                             //Check Subscribe ACK paket
                             CASE #tempMqttSubAckRcv OF
                               #NO_RESPONSE:  // Statement section case 1
                                 ;
                               #RESPONSE_GOOD:  // Statement section case 2 to 4
                                 //disable watchdog
                                 #statEnableTimerCommandWatchdog := FALSE;
                                 //Encoding done all sent
                                 #statPaketHeaderEncodeDone := FALSE;
                                 // Job done
                                 #statDone := TRUE;
                                 #statMqttCommandState := #MQTT_COMMAND_STATE_NO_PROCESSING;
                                 // Set Status back to connected
                                 #statStatus := #STATUS_JOB_EXECUTED;
                               #RESPONSE_PAKET_ID_INVALID:  // PaketId Invalid
                                 #statStatus := #ERR_MQTT_PAKET_ID_INVALID; // Set correct status that identifies error clearly
                                 #statSubfunctionStatus := #ERR_MQTT_PAKET_ID_INVALID; // Status or return value of called FBs, FCs and system blocks
                                 #statFBErrorState := #statFBState; // Set error state number for diagnostic 
                                 #statErrorAutoCleared := TRUE;
                                 #statMqttCommandState := #MQTT_COMMAND_STATE_NO_PROCESSING;
                               #RESPONSE_SUBSCRIBE_FAILED:
                                 #statStatus := #ERR_MQTT_SUBACK_FAILURE; // Set correct status that identifies error clearly
                                 #statSubfunctionStatus := #ERR_MQTT_SUBACK_FAILURE; // Status or return value of called FBs, FCs and system blocks
                                 #statFBErrorState := #statFBState; // Set error state number for diagnostic 
                                 #statErrorAutoCleared := TRUE;
                                 #statMqttCommandState := #MQTT_COMMAND_STATE_NO_PROCESSING;
                             END_CASE;
                           END_REGION SEND_SUBSCRIBE_WAIT_FOR_RESPONSE

                         #MQTT_COMMAND_STATE_BUILD_UNSUBSCRIBE:// Unsubscribe from topics
                           REGION UNSUBSCRIBE_FROM_TOPIC
                             //Remaining Length is the length of the variable header (PacketID, 2Bytes) plus the length of the Payload. 
                             //Max Len of Mqtt pakets is per Standard 268,435,455 Bytes (ff,ff,ff,7f)
                             //Calculate Remain Len will be
                             //Len of TOPIC   (max 3*16382 WChars= 49.146 Bytes)
                             //LenInfo Topic (2Byte)
                             //
                             //Set Status
                             #statStatus := #STATUS_MQTT_UNSUBSCRIBE;
                             // Must obey, if not currently sending PubAck Msg on a subscription
                             // Else, try in the next cycle
                             IF #tempTsendcBusy = FALSE // when tsendC is ready
                               AND #tempTsendcDone = FALSE // tsendC did not finish in this cycle
                               AND #statTsendcReq = FALSE // TsendC request was not already requested by pub ack msg
                             THEN
                               //Header not encoded
                               IF #statPaketHeaderEncodeDone = FALSE THEN
                                 //Init
                                 #statSendPaketTotalRemLen := 0;
                                 #statSendBufferPos := 0;
                                 #statUnsubscribeTopicEncodeState := #FIRST_ENCODING;
                                 #statUnsubscribeTopicPos := #FIRST_CHARACTER;
                                 #statUnsubscribeTopicLenUtf8Encoded := 0;
                                 #statPaketId += 1;//increment

                                 //check necessary boundaries

                                 IF LEN(#mqttTopic) = #LEN_NULL THEN
                                   #statStatus := #ERR_MQTT_COMMAND_UNSUBSCRIBE_TOPIC_INVALID; // Set correct status that identifies error clearly
                                   #statSubfunctionStatus := #ERR_MQTT_COMMAND_UNSUBSCRIBE_TOPIC_INVALID; // Status or return value of called FBs, FCs and system blocks
                                   #statFBErrorState := #statFBState; // Set error state number for diagnostic 
                                   #statErrorUserCleared := TRUE;
                                 ELSE // All ok
                                   //Add two Byte for Paket ID:
                                   #statSendPaketTotalRemLen := #statSendPaketTotalRemLen + #TWO_BYTE_LEN_INFO;
                                   //add unsubscribe  topic len
                                   FOR #tempLoopCounter := #FIRST_CHARACTER TO LEN(#mqttTopic) DO
                                     "LMQTT_ConvertToUtf8"(character     := #mqttTopic[#tempLoopCounter],
                                                           convertedUtf8 => #tempConvertedUtf8,
                                                           bytesUsed     => #tempBytesUsedUtf8,
                                                           error         => #tempErrorConvertUtf8,
                                                           status        => #tempStatusConvertUtf8);
                                     #statUnsubscribeTopicLenUtf8Encoded := #statUnsubscribeTopicLenUtf8Encoded + #tempBytesUsedUtf8;
                                   END_FOR;
                                   //Add len of topic plus len info
                                   #statSendPaketTotalRemLen := #statSendPaketTotalRemLen + #statUnsubscribeTopicLenUtf8Encoded + #TWO_BYTE_LEN_INFO;

                                   //Build Subscribe Telegram
                                   //Fixed Header - Write Paket Type
                                   #statSendBuffer[#statSendBufferPos] := #MQTT_MSG_TYPE_UNSUBSCRIBE;
                                   #statSendBufferPos += 1; // increment

                                   //Write Remaining Paket Len info 
                                   WHILE (#statSendPaketTotalRemLen > #DEFAULT_VALUE_ZERO)
                                   DO//See MQTT Spec for explanation of this calculation
                                     #statEncodedRemPaketLenAsByte := UDINT_TO_BYTE(#statSendPaketTotalRemLen MOD #SEND_LEN_MULTIPLIER_UDINT_128);
                                     #statSendPaketTotalRemLen := #statSendPaketTotalRemLen / #SEND_LEN_MULTIPLIER_UDINT_128;
                                     // if there are more data to encode, set the top bit of this byte
                                     IF #statSendPaketTotalRemLen > #DEFAULT_VALUE_ZERO
                                     THEN
                                       // Do this and continue while loop
                                       #statEncodedRemPaketLenAsByte := #statEncodedRemPaketLenAsByte OR UDINT_TO_BYTE(#SEND_LEN_MULTIPLIER_UDINT_128);
                                       #statSendBuffer[#statSendBufferPos] := #statEncodedRemPaketLenAsByte;
                                       #statSendBufferPos += 1;
                                     ELSE
                                       //do this and leave while loop
                                       #statSendBuffer[#statSendBufferPos] := #statEncodedRemPaketLenAsByte;
                                       #statSendBufferPos += 1;
                                     END_IF;
                                   END_WHILE;

                                   // Set Paket Id
                                   #tempWordForSliceAddress := UINT_TO_WORD(#statPaketId);
                                   #statSendBuffer[#statSendBufferPos] := #tempWordForSliceAddress.%B1; //MSB
                                   #statSendBufferPos += 1;
                                   #statSendBuffer[#statSendBufferPos] := #tempWordForSliceAddress.%B0; //LSB
                                   #statSendBufferPos += 1;

                                   //When all done, set encode to true
                                   #statPaketHeaderEncodeDone := TRUE;
                                 END_IF;
                               END_IF;

                               //Header Encoded - 
                               IF #statPaketHeaderEncodeDone = TRUE THEN
                                 //Unsubscribe Topic
                                 IF #statSendBufferPos <= #MAX_BUFFER_LEN_SEND - #TWO_BYTE_LEN_INFO THEN
                                   CASE #statUnsubscribeTopicEncodeState OF
                                     #FIRST_ENCODING:  // Statement section case 1
                                       //ADD len info into paket

                                       #tempWordForSliceAddress := UINT_TO_WORD(#statUnsubscribeTopicLenUtf8Encoded);
                                       #statSendBuffer[#statSendBufferPos] := #tempWordForSliceAddress.%B1; //MSB
                                       #statSendBufferPos += 1;
                                       #statSendBuffer[#statSendBufferPos] := #tempWordForSliceAddress.%B0; // LSB
                                       #statSendBufferPos += 1;

                                       FOR #tempLoopCounter := #statUnsubscribeTopicPos TO LEN(#mqttTopic) DO
                                         "LMQTT_ConvertToUtf8"(character     := #mqttTopic[#tempLoopCounter],
                                                               convertedUtf8 => #tempConvertedUtf8,
                                                               bytesUsed     => #tempBytesUsedUtf8,
                                                               error         => #tempErrorConvertUtf8,
                                                               status        => #tempStatusConvertUtf8);

                                         IF #statSendBufferPos + #tempBytesUsedUtf8 <= #MAX_BUFFER_LEN_SEND THEN
                                           #statUnsubscribeTopicPos += 1;
                                           CASE #tempBytesUsedUtf8 OF
                                             #UTF_1_BYTE_USED:  // Statement section case 1
                                               #statSendBuffer[#statSendBufferPos] := #tempConvertedUtf8.%B0;
                                               #statSendBufferPos += 1;
                                             #UTF_2_BYTE_USED:
                                               #statSendBuffer[#statSendBufferPos] := #tempConvertedUtf8.%B0;
                                               #statSendBufferPos += 1;
                                               #statSendBuffer[#statSendBufferPos] := #tempConvertedUtf8.%B1;
                                               #statSendBufferPos += 1;
                                             #UTF_3_BYTE_USED:  // Statement section case 2 to 4
                                               #statSendBuffer[#statSendBufferPos] := #tempConvertedUtf8.%B0;
                                               #statSendBufferPos += 1;
                                               #statSendBuffer[#statSendBufferPos] := #tempConvertedUtf8.%B1;
                                               #statSendBufferPos += 1;
                                               #statSendBuffer[#statSendBufferPos] := #tempConvertedUtf8.%B2;
                                               #statSendBufferPos += 1;
                                             ELSE  // Statement section ELSE
                                               ;
                                           END_CASE;
                                         ELSE
                                           //When buffer full
                                           #statUnsubscribeTopicEncodeState := #SUBSEQUENT_ENCODING;
                                           EXIT;
                                         END_IF;
                                       END_FOR;
                                       IF #statUnsubscribeTopicPos >= LEN(#mqttTopic) THEN
                                         #statUnsubscribeTopicEncodeState := #ENCODE_DONE;
                                       END_IF;

                                     #SUBSEQUENT_ENCODING:  // Statement section case 2 to 4
                                       FOR #tempLoopCounter := #statUnsubscribeTopicPos TO LEN(#mqttTopic) DO

                                         "LMQTT_ConvertToUtf8"(character     := #mqttTopic[#tempLoopCounter],
                                                               convertedUtf8 => #tempConvertedUtf8,
                                                               bytesUsed     => #tempBytesUsedUtf8,
                                                               error         => #tempErrorConvertUtf8,
                                                               status        => #tempStatusConvertUtf8);
                                         IF #statSendBufferPos + #tempBytesUsedUtf8 <= #MAX_BUFFER_LEN_SEND THEN
                                           #statUnsubscribeTopicPos += 1;
                                           CASE #tempBytesUsedUtf8 OF
                                             #UTF_1_BYTE_USED:  // Statement section case 1
                                               #statSendBuffer[#statSendBufferPos] := #tempConvertedUtf8.%B0;
                                               #statSendBufferPos += 1;
                                             #UTF_2_BYTE_USED:
                                               #statSendBuffer[#statSendBufferPos] := #tempConvertedUtf8.%B0;
                                               #statSendBufferPos += 1;
                                               #statSendBuffer[#statSendBufferPos] := #tempConvertedUtf8.%B1;
                                               #statSendBufferPos += 1;
                                             #UTF_3_BYTE_USED:  // Statement section case 2 to 4
                                               #statSendBuffer[#statSendBufferPos] := #tempConvertedUtf8.%B0;
                                               #statSendBufferPos += 1;
                                               #statSendBuffer[#statSendBufferPos] := #tempConvertedUtf8.%B1;
                                               #statSendBufferPos += 1;
                                               #statSendBuffer[#statSendBufferPos] := #tempConvertedUtf8.%B2;
                                               #statSendBufferPos += 1;
                                             ELSE  // Statement section ELSE
                                               ;
                                           END_CASE;
                                         ELSE
                                           //When buffer full
                                           EXIT;
                                         END_IF;
                                       END_FOR;
                                       IF #statUnsubscribeTopicPos >= LEN(#mqttTopic) THEN
                                         #statUnsubscribeTopicEncodeState := #ENCODE_DONE;
                                       END_IF;
                                     ELSE  // Skip when Done
                                       ;
                                   END_CASE;
                                 END_IF;

                                 //set Sendlen for TSendC Block
                                 #statTsendcLen := #statSendBufferPos; // Buffer pos equals amount of elements in send array
                                 //reset buffer pos
                                 #statSendBufferPos := 0;
                                 //enable Send Req
                                 #statTsendcReq := TRUE;
                                 //Set Watchdog
                                 #statEnableTimerCommandWatchdog := TRUE;
                                 //wait for send to be done
                                 #statMqttCommandState := #MQTT_COMMAND_STATE_SEND_UNSUBSCRIBE;
                               END_IF;
                             END_IF;
                           END_REGION UNSUBSCRIBE_FROM_TOPIC

                         #MQTT_COMMAND_STATE_SEND_UNSUBSCRIBE:
                           REGION SEND_UNSUBSCRIBE_WAIT_FOR_RESPONSE
                             //check tsend status
                             IF NOT #tempTsendcBusy AND #tempTsendcStatus = #TSENDC_JOB_DONE THEN
                               IF (#statUnsubscribeTopicEncodeState = #ENCODE_DONE) THEN
                                 //Encoding done all sent
                                 #statPaketHeaderEncodeDone := FALSE;
                               ELSE
                                 // More to Encode and send
                                 #statEnableTimerCommandWatchdog := FALSE;
                                 #statMqttCommandState := #MQTT_COMMAND_STATE_BUILD_UNSUBSCRIBE;
                               END_IF;
                             END_IF;
                             // Wait for timeout
                             IF #instTimerCommandWatchdog.Q THEN
                               #statEnableTimerCommandWatchdog := FALSE;
                               #statStatus := #ERR_MQTT_COMMAND_SEND_TIMEOUT; // Set correct status that identifies error clearly
                               #statSubfunctionStatus := #ERR_MQTT_COMMAND_SEND_TIMEOUT; // Status or return value of called FBs, FCs and system blocks
                               #statFBErrorState := #statFBState; // Set error state number for diagnostic 
                               #statErrorAutoCleared := TRUE;
                               #statMqttCommandState := #MQTT_COMMAND_STATE_NO_PROCESSING;
                             END_IF;
                             //Check Unsubscribe ACK paket
                             CASE #tempMqttUnSubAckRcv OF
                               #NO_RESPONSE:  // Statement section case 1
                                 ;
                               #RESPONSE_GOOD:  // Statement section case 2 to 4
                                 //disable watchdog
                                 #statEnableTimerCommandWatchdog := FALSE;
                                 //Encoding done all sent
                                 #statPaketHeaderEncodeDone := FALSE;
                                 // Job done
                                 #statDone := TRUE;
                                 #statMqttCommandState := #MQTT_COMMAND_STATE_NO_PROCESSING;
                                 // Set Status back to connected
                                 #statStatus := #STATUS_JOB_EXECUTED;
                               #RESPONSE_PAKET_ID_INVALID:
                                 #statStatus := #ERR_MQTT_PAKET_ID_INVALID; // Set correct status that identifies error clearly
                                 #statSubfunctionStatus := #ERR_MQTT_PAKET_ID_INVALID; // Status or return value of called FBs, FCs and system blocks
                                 #statFBErrorState := #statFBState; // Set error state number for diagnostic 
                                 #statErrorAutoCleared := TRUE;
                                 #statMqttCommandState := #MQTT_COMMAND_STATE_NO_PROCESSING;
                             END_CASE;
                           END_REGION SEND_UNSUBSCRIBE_WAIT_FOR_RESPONSE

                         #MQTT_COMMAND_STATE_SEND_PING:
                           REGION SEND_PING
                             //Set Status
                             #statStatus := #STATUS_MQTT_PING;
                             IF #tempTsendcBusy = FALSE // when tsendC is ready
                               AND #tempTsendcDone = FALSE // tsendC did not finish in this cycle
                               AND #statTsendcReq = FALSE // TsendC request was not already requested by pub ack msg
                             THEN
                               //Init
                               #statSendBufferPos := 0;
                               #statSendBuffer[#statSendBufferPos] := #MQTT_MSG_TYPE_PING;
                               #statSendBufferPos += 1;
                               //Remaining Lenght (must be 0)
                               #statSendBuffer[#statSendBufferPos] := 0;
                               #statSendBufferPos += 1;
                               #statTsendcLen := #statSendBufferPos;
                               //Start send request
                               #statTsendcReq := TRUE;
                               //Start watchdoc
                               #statEnableTimerCommandWatchdog := true;
                               //Next state
                               #statMqttCommandState := #MQTT_COMMAND_STATE_PING_RESP;
                             END_IF;
                           END_REGION MQTT_COMMAND_SEND_PING

                         #MQTT_COMMAND_STATE_PING_RESP:
                           REGION WAIT_FOR_PING_RESP
                             //Check, if Edge of Publish comes while ping
                             IF #tempCommandInput > 0 AND NOT #statCommandInputOld THEN
                               #statCommandInputBackup := #tempCommandInput;
                               #statCommandInputOld := true;
                             END_IF;
                             //check watchdog status
                             IF #instTimerCommandWatchdog.Q THEN
                               #statEnableTimerCommandWatchdog := FALSE;
                               #statStatus := #ERR_MQTT_COMMAND_SEND_TIMEOUT; // Set correct status that identifies error clearly
                               #statSubfunctionStatus := #ERR_MQTT_COMMAND_SEND_TIMEOUT; // Status or return value of called FBs, FCs and system blocks
                               #statFBErrorState := #statFBState; // Set error state number for diagnostic 
                               #statErrorAutoCleared := TRUE;
                               #statMqttCommandState := #MQTT_COMMAND_STATE_NO_PROCESSING;
                             END_IF;
                             //Check PingRsp paket
                             CASE #tempMqttPingRspRcv OF
                               #NO_RESPONSE:  // Statement section case 1
                                 ;
                               #RESPONSE_GOOD:
                                 //disable watchdog
                                 #statEnableTimerCommandWatchdog := FALSE;
                                 //Go to no processing
                                 #statMqttCommandState := #MQTT_COMMAND_STATE_NO_PROCESSING;
                                 //set Status
                                 #statStatus := #STATUS_MQTT_CONNECTED;
                                 IF #statCommandInputBackup <> 0 THEN
                                   #statMqttCommandState := BYTE_TO_DINT(#statCommandInputBackup);
                                   #statCommandInputBackup := 0;
                                   #statCommandInputOld := false;
                                 END_IF;
                             END_CASE;
                           END_REGION MQTT_COMMAND_PING_RESP
                         ELSE  // Statement section ELSE
                           REGION ERROR_MULTIPLE_INPUT
                             #statMqttCommandState := #MQTT_COMMAND_STATE_NO_PROCESSING; // reset back to idle
                             #statStatus := #ERR_MQTT_COMMAND_MULTIPLE_INPUT; // Set correct status that identifies error clearly
                             #statSubfunctionStatus := #ERR_MQTT_COMMAND_MULTIPLE_INPUT; // Status or return value of called FBs, FCs and system blocks
                             #statFBErrorState := #statFBState; // Set error state number for diagnostic 
                             #statErrorAutoCleared := TRUE;
                           END_REGION ERROR_MULTIPLE_INPUT 
                       END_CASE;
                     END_REGION

                     REGION CHECK_PING_TIMER
                       //If no job is running check if keepalive experied
                       IF #statMqttCommandState = #MQTT_COMMAND_STATE_NO_PROCESSING
                         AND #instMqttKeepAliveTimer.Q THEN
                         //reset the timer
                         RESET_TIMER(#instMqttKeepAliveTimer);
                         //go to ping state
                         #statMqttCommandState := #MQTT_COMMAND_STATE_SEND_PING;
                       END_IF;
                     END_REGION CHECK_PING_TIMER

                     //Edge detection "publish / subscribe/unsubscribe" input
                     #statPublishOld := #tempPublish;
                     #statSubscribeOld := #tempSubscribe;
                     #statUnsubscribeOld := #tempUnsubscribe;
                   END_REGION CONNECTED

                 ELSE   // Undefined state in state machine reached
                   #statStatus := #ERR_UNDEFINED_STATE;
                   #statErrorUserCleared := TRUE;
               END_CASE;

             END_REGION MQTT_STATE_MACHINE
           END_IF;
         END_REGION FB_OPERATING_MONITOR_TCP

       #FB_STATE_TCP_RECONNECTING:
         REGION FB_STATE_TCP_RECONNECTING
           IF #tempTsendcStatus = #TSENDC_EST_OK THEN
             #statErrorAutoCleared := FALSE;
             // Update edge detection
             #statPublishOld := #tempPublish;
             #statSubscribeOld := #tempSubscribe;
             #statUnsubscribeOld := #tempUnsubscribe;
             //Monitor Connection
             #statFBState := #FB_STATE_OPERATING_MONITOR_TCP;
             // Begin MQTT Connection
             #statMqttConnectState := #MQTT_CONNECT_STATE_BUILD_PAKET;
           END_IF;
         END_REGION FB_STATE_TCP_RECONNECTING
       #FB_STATE_DISABLING: // Disabling active
         REGION DISABLING FB
           //  Disabling, e.g. closing connections, etc.
           // When disabling is complete the bit #statDisablingCompleted must be set
           // When MQTT is connected, send disconnect
           IF #statMqttConnectState = #MQTT_CONNECT_STATE_CONNECTED THEN
             IF #statTsendcReq = TRUE THEN
               //Interrupt any existing send jobs
               #statTsendcReq := FALSE;
             ELSE
               // INIT
               #statSendBufferPos := 0;
               //Build fixed Header
               //Message Type
               #statSendBuffer[#statSendBufferPos] := #MQTT_MSG_TYPE_DISCONNECT;
               #statSendBufferPos += 1;
               //Remaining Length (must be O)
               #statSendBuffer[#statSendBufferPos] := #REMAINIG_LEN_0;
               #statSendBufferPos += 1;
               //send request
               #statTsendcLen := #statSendBufferPos;
               #statTsendcReq := TRUE;
               #statMqttConnectState := #MQTT_CONNECT_STATE_DISCONNECTED;
             END_IF;
           ELSE
             //Disable TCP Connection
             #statTsendcReq := FALSE;
             #statTsendcEnable := FALSE;
             #statEnableTimerCommandWatchdog := TRUE;
           END_IF;
           // When TCP connection is closed
           IF #tempTsendcStatus = #TSENDC_DISCONNECTED THEN
             #statEnableTimerCommandWatchdog := FALSE;
             #statDisablingCompleted := TRUE;
           ELSIF #instTimerCommandWatchdog.Q THEN
             #statEnableTimerCommandWatchdog := FALSE;
             #statDisablingCompleted := TRUE;
           END_IF;
         END_REGION DISABLING FB
       ELSE // Undefined state in state machine reached
         #statStatus := #ERR_UNDEFINED_STATE;
         #statErrorUserCleared := TRUE;
     END_CASE;
   END_REGION STATE_MACHINE

   REGION OUTPUTS
     // Write outputs
     IF (#statDisablingCompleted = TRUE) THEN
       // Reset outputs if disabling completed
       #statValid := FALSE;
       #statBusy := FALSE;
       #statError := FALSE;
       #statDone := FALSE;
       #statErrorUserCleared := FALSE;
       #statErrorAutoCleared := FALSE;
       #statStatus := #STATUS_NO_CALL;
       // Reset application specific outputs
       #statRcvMsgStatus := #MSG_DECODE_STATUS_NO_NEW_MSG;
       #statRcvMsgDataLen := 0;

     ELSIF (#statErrorUserCleared = TRUE) AND (#statError = FALSE) THEN
       // Error can only be cleared by user; rising edge at enable input is needed to continue 
       #statValid := FALSE;
       #statBusy := FALSE;
       #statDone := FALSE;
       #statError := TRUE;
       // Write diagnostics
       #diagnostics.status := #statStatus;
       #diagnostics.subfunctionStatus := #statSubfunctionStatus;
       #diagnostics.stateNumber := #statFBErrorState;
       // execution aborted --> set state no processing
       #statTsendcEnable := FALSE; // Terminate Connection, no reason keep it up.
       #statFBState := #FB_STATE_NO_PROCESSING;
       #statMqttConnectState := #MQTT_CONNECT_STATE_NO_PROCESSING;
       #statMqttCommandState := #MQTT_COMMAND_STATE_NO_PROCESSING;
       #statRcvMsgDecodeState := #MSG_DECODE_STATE_NO_PROCESSING;

     ELSIF (#statErrorAutoCleared = TRUE) AND (#statError = FALSE) THEN
       // Error can be reset by FB automatically
       #statValid := FALSE;
       #statBusy := TRUE;
       #statError := TRUE;
       #statDone := FALSE;

       // Write diagnostics
       #diagnostics.status := #statStatus;
       #diagnostics.subfunctionStatus := #statSubfunctionStatus;
       #diagnostics.stateNumber := #statFBErrorState;
       // Handling of autocleared error
       CASE #statStatus OF
           //Just signal error and reset autocleared error afterwards.
         #ERR_MQTT_PAKET_ID_INVALID, #ERR_MQTT_SUBACK_FAILURE, #ERR_MQTT_CONNECT_TIMEOUT,
         #ERR_MQTT_COMMAND_SEND_TIMEOUT, #ERR_MQTT_COMMAND_MULTIPLE_INPUT, #ERR_CNT_EXCEEDS_ARRAY_DIMENSION,
         #ERR_MQTT_COMMAND_PUBLISH_TOPIC_INVALID, #ERR_QOS_INVALID, #ERR_MQTT_COMMAND_SUBSCRIBE_TOPIC_INVALID:
           #statErrorAutoCleared := FALSE;

         ELSE  // Statement section ELSE
           ;
       END_CASE;

     ELSIF (#statErrorAutoCleared = FALSE) AND (#statErrorUserCleared = FALSE) AND (#statError = TRUE) THEN
       // If autocleared error is acknowledged
       #statValid := TRUE;
       #statBusy := TRUE;
       #statError := FALSE;
       #statDone := FALSE;

       //   this line  more detailed status information is used instead of "#STATUS_SUBSEQUENT_CALL"
       CASE #statStatus OF
         #ERR_TCP_RECONNECTING, #ERR_MQTT_CONNECT_TIMEOUT:  // Reconnecting ok, start Mqtt reconnnect
           //set status
           #statStatus := #STATUS_MQTT_CONNECTING;
           //in the following status codes status stays connected. 
         #ERR_MQTT_PAKET_ID_INVALID, #ERR_MQTT_SUBACK_FAILURE, #ERR_MQTT_COMMAND_SEND_TIMEOUT,
         #ERR_MQTT_COMMAND_MULTIPLE_INPUT, #ERR_CNT_EXCEEDS_ARRAY_DIMENSION, #ERR_MQTT_COMMAND_PUBLISH_TOPIC_INVALID,
         #ERR_QOS_INVALID, #ERR_MQTT_COMMAND_SUBSCRIBE_TOPIC_INVALID:
           #statStatus := #STATUS_MQTT_CONNECTED;
         ELSE  // Statement section ELSE
           ;
       END_CASE;
     END_IF;

     // Write static values to outputs
     #valid := #statValid;
     #busy := #statBusy;
     #error := #statError;
     #status := #statStatus;
     //block sets ENO automatically:
     //ENO := TRUE;
     //Write application specific static values to outputs
     #done := #statDone;
     #receivedMsgStatus := #statRcvMsgStatus;
     #receivedMsgDataLen := #statRcvMsgDataLen;
   END_REGION OUTPUTS
END_FUNCTION_BLOCK

// folder: LMQTT/Utilities

FUNCTION "LMQTT_ConvertToUtf8" : Void   // FC6, SCL
TITLE = LMQTT_ConvertToUtf8
{ S7_Optimized_Access := 'TRUE' }
AUTHOR : SIEMENS
FAMILY : LMQTT
VERSION : 1.0
// Function to convert a WCHAR to a UTF-8 conformant byte sequence
   VAR_INPUT
      character : WChar;   // Character that shall be converted to UTF-8
   END_VAR
   VAR_OUTPUT
      convertedUtf8 : DWord;   // UTF-8 conformant byte sequence. B0 stores first Byte, B1 second and B2 third Byte. B3 is not used
      bytesUsed : USInt;   // Amount of Bytes converted. Ranges from 1 to 3.
      error : Bool;   // TRUE: An error occurred during the execution of the FC
      status : Word;   // 16#0000 - 16#7FFF: Status of the FC, 16#8000 - 16#FFFF: Error identification
   END_VAR
   VAR_TEMP
      tempStatus : Word;   // temp value for output 'status'
      tempConvertedUtf8 : DWord;   // temp value for output 'convertedUtf8'
      tempBytesUsed : USInt;   // temp value for output 'bytesUsed'
      tempCharacter : WChar;   // temp value for input 'character'
   END_VAR
   // Ret_Val : No return for this FC - see error and status output
   VAR CONSTANT
      STATUS_NO_ERROR : Word := 16#0000;   // no error status
      STATUS_EXECUTION_FINISHED : Word := 16#0000;   // Execution finished without errors
      ERR_UNDEFINED : Word := 16#8000;   // Error due to an undefined case
      USINT_NULL : USInt := 0;   // Init value with 0
      DWORD_NULL : DWord := 16#0000_0000;   // Init value with 0
      EMPTY_WCHAR : WChar := WCHAR#' ';   // Empty WChar for comparison
      BELOW_7F : Word := 16#007F;   // Upper limit for character if only one Byte used
      BELOW_7FF : Word := 16#07FF;   // Upper limit for character if two Byte used
      BELOW_MAX_FFFF : Word := 16#FFFF;   // Upper limit for character if three Byte used
      BYTE_3F : Byte := 16#3F;   // Conversion Value
      BYTE_80 : Byte := 16#80;   // Conversion Value
      BYTE_C0 : Byte := 16#C0;   // Conversion Value
      BYTE_E0 : Byte := 16#E0;   // Conversion Value
      USINT_ONE : USInt := 1;   // Const Value to assign amount of bytes used
      USINT_TWO : USInt := 2;   // Const Value to assign amount of bytes used
      USINT_THREE : USInt := 3;   // Const Value to assign amount of bytes used
   END_VAR
BEGIN
   REGION BLOCK INFO HEADER
       //=============================================================================
       // SIEMENS AG
       // (c)Copyright 2020
       //-----------------------------------------------------------------------------
       // Library:       LMQTT
       // Tested with:   CPU 1516-3 PN/DP V2.8
       // Engineering:   TIA Portal V16
       // Restrictions:  --
       // Requirements:  --
       // Functionality: Converts a single WChar Character to a valid UTF-8 encoded byte sequence and saves this to a DWord.
       //                The amount of bytes saved is stored in bytesUsed Output.
       //-----------------------------------------------------------------------------
       // Change log table:
       // Version    Date         Expert in charge         Changes applied
       // 03.00.00   01.10.2020   Siemens Online Support   First released version
       //=============================================================================
   END_REGION

   REGION INITIALISATION  
       // Initialize functionality: reset of variables, diagnostics, etc.
       #tempConvertedUtf8 := #DWORD_NULL;
       #tempBytesUsed := #USINT_NULL;
       #tempStatus := #STATUS_NO_ERROR;
       //assign temp value from input:
        #tempCharacter := #character;

   END_REGION

   REGION PROGRAM LOGIC
       // Use this region for application specific code
       IF #tempCharacter = #EMPTY_WCHAR THEN
           //will be only 1 byte occupied
           #tempConvertedUtf8 := WCHAR_TO_DWORD(#tempCharacter);
           #tempBytesUsed := #USINT_ONE;
       ELSIF (WCHAR_TO_WORD(#tempCharacter) <= (#BELOW_7F)) THEN
           //will be only 1 byte occupied
           #tempConvertedUtf8 := WCHAR_TO_DWORD(#tempCharacter);
           #tempBytesUsed := #USINT_ONE;
       ELSIF (WCHAR_TO_WORD(#tempCharacter) <= (#BELOW_7FF)) THEN
           //will be 2 byte occupied
           #tempConvertedUtf8.%B1 := (WCHAR_TO_BYTE(#tempCharacter) AND #BYTE_3F) OR #BYTE_80;
           #tempConvertedUtf8.%B0 := WORD_TO_BYTE(SHR(IN := WCHAR_TO_WORD(#tempCharacter), N := 6)) OR #BYTE_C0;
           #tempBytesUsed := #USINT_TWO;
       ELSIF (WCHAR_TO_WORD(#tempCharacter) <= (#BELOW_MAX_FFFF)) THEN
           //will be 3 byte occupied
           #tempConvertedUtf8.%B2 := (WCHAR_TO_BYTE(#tempCharacter) AND #BYTE_3F) OR #BYTE_80;
           #tempConvertedUtf8.%B1 := (WORD_TO_BYTE(SHR(IN := WCHAR_TO_WORD(#tempCharacter), N := 6)) AND #BYTE_3F) OR #BYTE_80;
           #tempConvertedUtf8.%B0 := WORD_TO_BYTE(SHR(IN := WCHAR_TO_WORD(#tempCharacter), N := 12)) OR #BYTE_E0;
           #tempBytesUsed := #USINT_THREE;
       END_IF;
   END_REGION

   REGION OUTPUTS
       // Write application specific temp values to outputs
       #bytesUsed := #tempBytesUsed;
       #convertedUtf8 := #tempConvertedUtf8;
       // Write error and status
       #error := #tempStatus.%X15;
       #status := #tempStatus;
       // ENO mechanism is not used --> ENO := TRUE;
       ENO := TRUE;
   END_REGION
END_FUNCTION

// ===== PLC "PLC_1500"  CPU 1516-3 PN/DP =====

TYPE "crossroad_input"
   STRUCT
      CrossroadType : Bool;
      btnCrossroadStart : Bool;
      btnCrossroadPause : Bool;
      btnCrossroadStop : Bool;
      btnCrosswalk1 : Bool;
      btnCrosswalk2 : Bool;
   END_STRUCT;
END_TYPE

TYPE "crossroad_output"
   STRUCT
      traffic_light1_green : Bool;
      traffic_light1_yellow : Bool;
      traffic_light1_red : Bool;
      traffic_light2_green : Bool;
      traffic_light2_yellow : Bool;
      traffic_light2_red : Bool;
      pedestrian_light1_green : Bool;
      pedestrian_light1_red : Bool;
      pedestrian_light2_green : Bool;
      pedestrian_light2_red : Bool;
   END_STRUCT;
END_TYPE

TYPE "crossroad_internal"
   STRUCT
      CTU_reset : Bool;
      CTU_current_value : Int;
      Day_Sequence : Int;
      Night_Sequence : Int;
      Off : Bool;
   END_STRUCT;
END_TYPE

// folder: Common

TYPE "typeDiagnostics"
TITLE = typeDiagnostics
// Provides a structure for detailed diagnostics
   STRUCT
      status : Word;   // Status of the block or error identification when error occurred
      subfunctionStatus : DWord;   // Status or return value of called FBs, FCs and system blocks
      stateNumber : DInt;   // State in the state machine of the block where the error occurred
   END_STRUCT;
END_TYPE

// folder: LHTTP

TYPE "LHTTP_typeTLS"
   STRUCT
      validateServerIdentity : Bool;   // Validate the subjectAlternateName in the X.509-V3 certificate of the server to check the identity of the server
      serverCert : UDInt;   // ID of the X.509-V3 certificate (usually a CA certificate) that is used by the TLS client to validate the TLS server authentication. If this parameter is 0, the TLS client uses all (CA) certificates currently loaded in the client certificate store to validate the server authentication.
      clientCert : UDInt;   // ID of own X.509 V3 certificate
   END_STRUCT;
END_TYPE

// folder: LMQTT

TYPE "LMQTT_typeConnParam"
TITLE = LMQTT_typeConnParams
// Specifies connection parameters for the mqtt connection
   STRUCT
      hwId : Hw_Any;   // Hardware identifier of the interface. 0: interface is selected automatically
      connId : Conn_Ouc := 1;   // Unique connection identifier (1..4095)
      broker : String;   // Hostname or IP address of broker
      port : UInt := 1883;   // Port on the broker
      tls : Struct   // Parameters for TLS encryption
         enableTls : Bool;   // TRUE: Enables TLS, FALSE: disable TLS
         validateServerIdentity : Bool;   // TRUE: Validate server certificate, FALSE: No validation of server certificate
         brokerCert : UDInt;   // ID of the broker's certificate in TIA Portal
         clientCert : UDInt;   // ID of the client's certificate in TIA Portal
      END_STRUCT;
      keepAlive : UInt;   // Keepalive mechanism for MQTT in seconds. 0: disabled.
   END_STRUCT;
END_TYPE

// folder: Communication/RESTAPI

DATA_BLOCK "RESTAPI_variables"   // DB9
{ S7_Optimized_Access := 'TRUE' }
VERSION : 0.1
   VAR
      server_url : String := 'http://localhost:5000/api/data';
      "time" : Time := T#50ms;
      contentType : String := 'application/json';
      databody : String;
      execute_get : String;
      execute_post : Bool;
      headerbase : String;
      requestpaylod : String;
      countheader : USInt;
      responseData_get : Array[0..1000] of Char;
      responseData_post : Array[0..1000] of Char;
      header : Array[0..255] of Char;
   END_VAR
BEGIN
END_DATA_BLOCK

DATA_BLOCK "LHTTP_Get_DB"   // DB10
{ S7_Optimized_Access := 'TRUE' }
AUTHOR : Siemens Industry Online Support
FAMILY : LHTTP
VERSION : 2.2
// stored: InstanceOfName LHTTP_Get
"LHTTP_Get"
BEGIN
END_DATA_BLOCK

DATA_BLOCK "LHTTP_PostPut_DB"   // DB11
{ S7_Optimized_Access := 'TRUE' }
AUTHOR : Siemens Industry Online Support
FAMILY : LHTTP
VERSION : 2.2
// stored: InstanceOfName LHTTP_PostPut
"LHTTP_PostPut"
BEGIN
END_DATA_BLOCK

// folder: crossroad

DATA_BLOCK "CrosswalkDataDB"   // DB6
{ S7_Optimized_Access := 'FALSE' }
VERSION : 0.1
   VAR
      inputs : "crossroad_input";
      outputs : "crossroad_output";
      internal : "crossroad_internal";
   END_VAR
BEGIN
END_DATA_BLOCK

// folder: (top level)

ORGANIZATION_BLOCK "Main"   // OB1, LAD, ProgramCycle
TITLE = "Main Program Sweep (Cycle)"
{ S7_Optimized_Access := 'TRUE' }
VERSION : 0.1
   VAR_INPUT
      Initial_Call : Bool;   // Initial call of this OB
      Remanence : Bool;   // =True, if remanent data are available
   END_VAR
BEGIN
END_ORGANIZATION_BLOCK

ORGANIZATION_BLOCK "CyclicInterrupt"   // OB30, LAD, CyclicInterrupt
{ S7_Optimized_Access := 'TRUE' }
VERSION : 0.1
   VAR_INPUT
      Initial_Call : Bool;   // Initial call of this OB
      Event_Count : Int;   // Events discarded
   END_VAR
BEGIN
END_ORGANIZATION_BLOCK

ORGANIZATION_BLOCK "Startup"   // OB100, SCL, Startup
TITLE = "Complete Restart"
{ S7_Optimized_Access := 'TRUE' }
VERSION : 0.1
   VAR_INPUT
      LostRetentive : Bool;   // True if retentive data are lost
      LostRTC : Bool;   // True if date and time are lost
   END_VAR
BEGIN
END_ORGANIZATION_BLOCK

// folder: Communication/Modbus

FUNCTION "Modbus_Server" : Void   // FC3, LAD
{ S7_Optimized_Access := 'TRUE' }
VERSION : 0.1
BEGIN

REGION Network 1
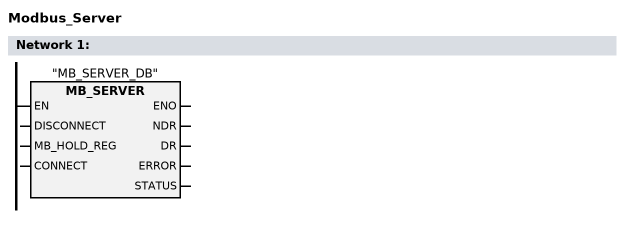
   "MB_SERVER_DB"();   // MB_SERVER
END_REGION
END_FUNCTION

FUNCTION "Modbus_Klient" : Void   // FC4, LAD
{ S7_Optimized_Access := 'TRUE' }
VERSION : 0.1
BEGIN

REGION Network 1
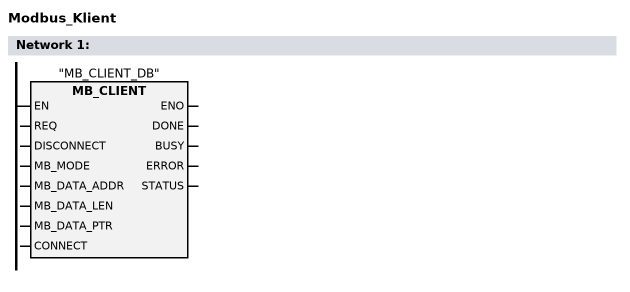
   "MB_CLIENT_DB"();   // MB_CLIENT
END_REGION
END_FUNCTION

// folder: Communication/RESTAPI

FUNCTION_BLOCK "RESTAPI_com"   // FB1, LAD
{ S7_Optimized_Access := 'TRUE' }
VERSION : 0.1
   VAR
      valueBtnCrossroadStart : String;
      valueBtnCrossroadPause : String;
      valueBtnCrossroadStop : String;
      valueBtnCrosswalk1 : String;
      valueBtnCrosswalk2 : String;
      valueCrossroadType : String;
      valueTrafficLight1_green : String;
      valueTrafficLight1_yellow : String;
      valueTrafficLight1_red : String;
      tmpBody : String;
   END_VAR
BEGIN

REGION Network 1 (SCL)
   //"RESTAPI_variables".databody := '{"mission_id": "fb2436de-1545-11f0-8560-000e8e9851ad"}';

   IF "CrosswalkDataDB".outputs.traffic_light1_green THEN
       #valueTrafficLight1_green := '"true"';
   ELSE
       #valueTrafficLight1_green := '"false"';
   END_IF;

   IF "CrosswalkDataDB".outputs.traffic_light1_yellow THEN
       #valueTrafficLight1_yellow := '"true"';
   ELSE
       #valueTrafficLight1_yellow := '"false"';
   END_IF;

   #tmpBody := CONCAT(IN1 := '{"trafficLights1_green": ', IN2 := #valueTrafficLight1_green);
   #tmpBody := CONCAT(IN1 := #tmpBody, IN2 := ', "trafficLights1_yellow": ');


   "RESTAPI_variables".databody := CONCAT(IN1 := #tmpBody,IN2 := '}');
END_REGION

REGION Network 2: Loop for writting to server
   // Loop for writting to server: 
   // - lights
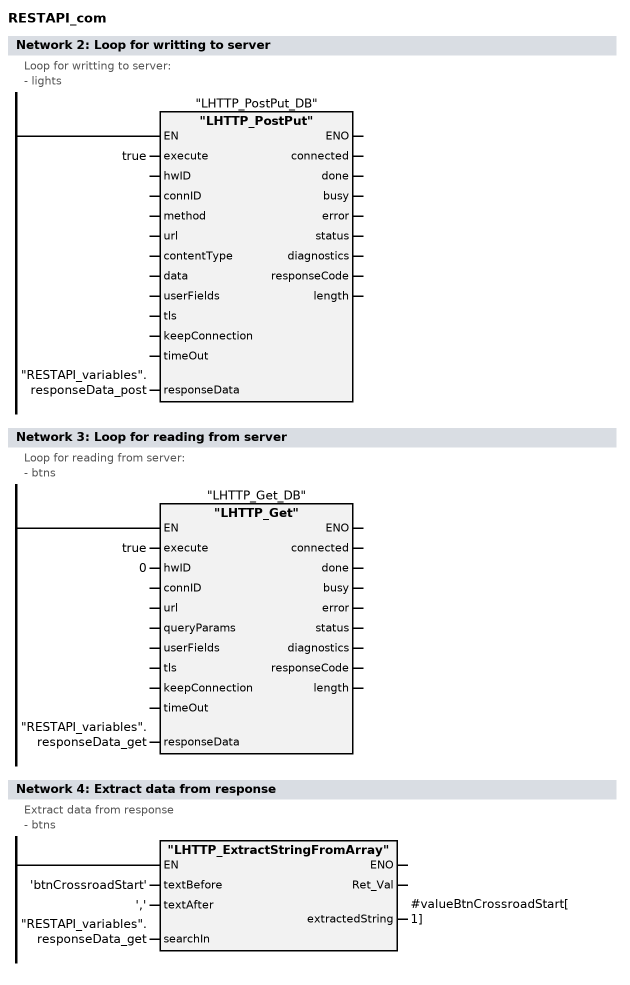
   RUNG wire#powerrail
      "LHTTP_PostPut_DB"(execute := true, hwID :=, connID :=, method :=, url :=, contentType :=, data :=, userFields :=, tls :=, keepConnection :=, timeOut :=, responseData := "RESTAPI_variables".responseData_post, connected =>, done =>, busy =>, error =>, status =>, diagnostics =>, responseCode =>, length =>)
   END_RUNG
   // the same network as SCL:
   "LHTTP_PostPut_DB"(execute := true, responseData := "RESTAPI_variables".responseData_post);   // "LHTTP_PostPut"
END_REGION

REGION Network 3: Loop for reading from server
   // Loop for reading from server:
   // - btns
   RUNG wire#powerrail
      "LHTTP_Get_DB"(execute := true, hwID := 0, connID :=, url :=, queryParams :=, userFields :=, tls :=, keepConnection :=, timeOut :=, responseData := "RESTAPI_variables".responseData_get, connected =>, done =>, busy =>, error =>, status =>, diagnostics =>, responseCode =>, length =>)
   END_RUNG
   // the same network as SCL:
   "LHTTP_Get_DB"(execute := true, hwID := 0, responseData := "RESTAPI_variables".responseData_get);   // "LHTTP_Get"
END_REGION

REGION Network 4: Extract data from response
   // Extract data from response 
   // - btns
   RUNG wire#powerrail
      "LHTTP_ExtractStringFromArray"(textBefore := 'btnCrossroadStart', textAfter := ',', searchIn := "RESTAPI_variables".responseData_get, Ret_Val =>, extractedString => #valueBtnCrossroadStart[1])
   END_RUNG
   // the same network as SCL:
   "LHTTP_ExtractStringFromArray"(textBefore := 'btnCrossroadStart',
                           textAfter := ',',
                           searchIn := "RESTAPI_variables".responseData_get,
                           extractedString => #valueBtnCrossroadStart[1]);
END_REGION
END_FUNCTION_BLOCK

// folder: Communication/S7

FUNCTION "S7_com" : Void   // FC7, LAD
{ S7_Optimized_Access := 'TRUE' }
VERSION : 0.1
BEGIN

REGION Network 1
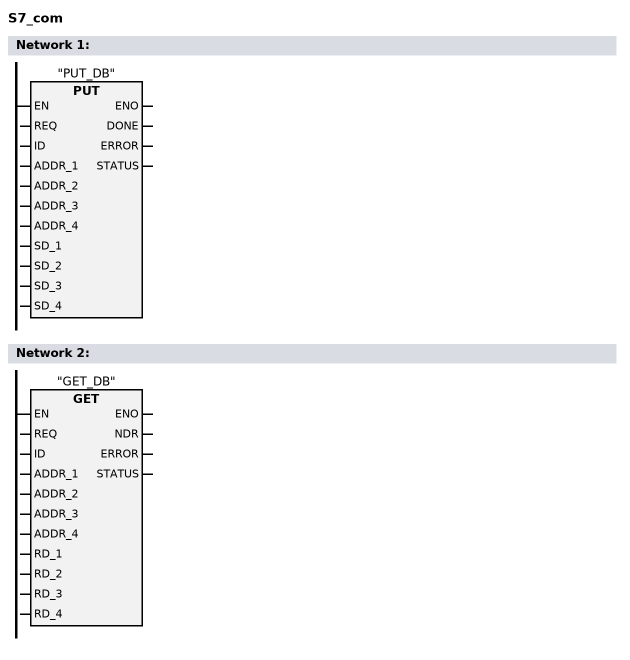
   "PUT_DB"();   // PUT
END_REGION

REGION Network 2
   "GET_DB"();   // GET
END_REGION
END_FUNCTION

// folder: Communication/TCPIP

FUNCTION "TCPIP" : Void   // FC2, LAD
{ S7_Optimized_Access := 'TRUE' }
VERSION : 0.1
BEGIN

REGION Network 1: Klient (PLC) -> Server (C#)
   // Klient složí zprávu o stavu světel. Pošle ji na server (TSEND). Server očekává zprávu o stavu tlačítek (TRCV). Po obdržení zprávy updatuje tlačítka.
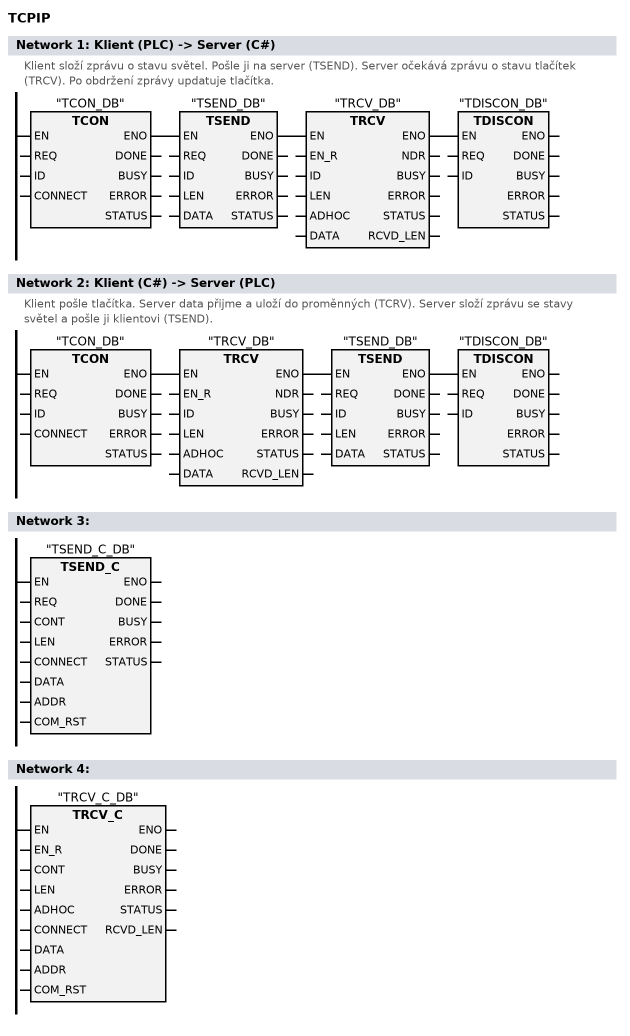
   // ENO of a box is taken as its EN; it also drops when the box reports an error
   "TCON_DB"();   // TCON
   "TSEND_DB"();   // TSEND
   "TRCV_DB"();   // TRCV
   "TDISCON_DB"();   // TDISCON
END_REGION

REGION Network 2: Klient (C#) -> Server (PLC)
   // Klient pošle tlačítka. Server data přijme a uloží do proměnných (TCRV). Server složí zprávu se stavy světel a pošle ji klientovi (TSEND).
   // ENO of a box is taken as its EN; it also drops when the box reports an error
   "TCON_DB"();   // TCON
   "TRCV_DB"();   // TRCV
   "TSEND_DB"();   // TSEND
   "TDISCON_DB"();   // TDISCON
END_REGION

REGION Network 3
   "TSEND_C_DB"();   // TSEND_C
END_REGION

REGION Network 4
   "TRCV_C_DB"();   // TRCV_C
END_REGION
END_FUNCTION

// folder: Libraries/Common

FUNCTION "IsIPAddress" : Bool   // FC1, SCL
TITLE = IsIPAddress
{ S7_Optimized_Access := 'TRUE' }
VERSION : 0.1
// Evaluates whether a given String contains a valid IP address
   VAR_INPUT
      address : String;   // Address to be evaluated
   END_VAR
   VAR_OUTPUT
      ipAddress : IP_V4;   // Parsed IP address if passed address is IP address
   END_VAR
   VAR_TEMP
      tempAddress : String;   // Passed address
      tempOctet : String;   // Current octet
      tempIndex : DInt;   // Index for loop
      tempPos : Int;   // Position of found separator
      tempNum : Int;   // Converted octet
      tempIp : IP_V4;   // Parsed IP address
   END_VAR
   // Ret_Val : Return value
   VAR CONSTANT
      MAX_VALUE : USInt := 255;   // Max. valid value of octet
      NUM_OCTETS : DInt := 4;   // Number of octets
      CHAR_ZERO : Char := '0';   // ASCII character '0'
   END_VAR
BEGIN
   REGION BLOCK INFO HEADER
     //===============================================================================
     // SIEMENS / (c)Copyright 2024
     //-------------------------------------------------------------------------------
     // Title:        IsIPAddress
     // Function:     Evaluates whether a given String contains a valid IP address
     // Library:      --
     // Author:       Siemens Industry Online Support
     // Tested with:  CPU 1515-2 PN V3.1
     // Engineering:  TIA Portal V17
     // Restrictions: --
     // Requirements: S7-1200 with firmware V4.4 or higher
     //               S7-1500 with firmware V2.0 or higher
     //-------------------------------------------------------------------------------
     // Change log table:
     // Version  | Date       | Expert in charge       | Changes applied
     //-------------------------------------------------------------------------------
     // 01.00.00 | 2024-02-12 | Online Support         | First released version
     //===============================================================================
   END_REGION

   #tempAddress := #address;
   #IsIPAddress := FALSE; // Will be overwritten if IP address is detected
   #ipAddress := #tempIp; // Zero output parameter

   FOR #tempIndex := 1 TO #NUM_OCTETS DO
     #tempPos := FIND(IN1 := #tempAddress, IN2 := '.'); // Find separator

     IF (#tempPos > 0 OR #tempIndex = #NUM_OCTETS) // Separator found with exception of last octet
       AND NOT (#tempPos > 0 AND #tempIndex = #NUM_OCTETS) // No separator found in last octet
       AND #tempPos <= 4 // 3  characters or less
     THEN
       IF #tempIndex < #NUM_OCTETS THEN // First three octets
         #tempOctet := LEFT(IN := #tempAddress, L := #tempPos - 1);
       ELSE// Last octet
         #tempOctet := #tempAddress;
       END_IF;

       STRG_VAL(IN := #tempOctet,
                FORMAT := 0,
                P := 1,
                OUT => #tempNum);

       IF #tempNum >= 0 AND #tempNum <= #MAX_VALUE // Within 0 and 255
         AND NOT (#tempNum = 0 AND #tempIndex = 1) // Not 0 in first octet
         AND NOT (#tempNum = 0 AND #tempOctet[1] <> #CHAR_ZERO) // Not 0 because of invalid character
       THEN
         #tempIp.ADDR[#tempIndex] := INT_TO_BYTE(#tempNum);
         #tempAddress := RIGHT(IN := #tempAddress, L := LEN(#tempAddress) - #tempPos); // Remove evaluated octet
       ELSE // Address is not IP address
         EXIT;
       END_IF;
     ELSE // Address is not IP address
       EXIT;
     END_IF;

     IF #tempIndex = #NUM_OCTETS THEN // End of loop reached, address is IP address
       #ipAddress := #tempIp;
       #IsIPAddress := true;
     END_IF;
   END_FOR;
END_FUNCTION

// folder: Libraries/LHTTP

FUNCTION_BLOCK "LHTTP_Get"   // FB8, SCL
TITLE = LHTTP_Get
{ S7_Optimized_Access := 'TRUE' }
AUTHOR : Siemens Industry Online Support
FAMILY : LHTTP
VERSION : 2.2
// Implements the HTTP GET method
   VAR_INPUT
      execute : Bool;   // Send HTTP request
      hwID : Hw_Any;   // Hardware ID of Ethernet interface
      connID : Conn_Ouc := 1;   // Unique connection ID
      url : String;   // URL, i.e. "http://www.siemens.com/simatic"
      queryParams : String;   // Additional query parameters if "url" is not long enough, i.e. "lang=en&q=simatic"; "?" or "&" is inserted automatically in between "url" and "queryParameters". / Optional query parameters that are appended to URL, i.e. "lang=en&q=simatic"
      userFields : Array[0..#UPPER_USER_FIELDS] of Char;   // Additional user-defined header fields
      tls : "LHTTP_typeTLS";   // TLS certificates for secure connections (HTTPS), leave open for non-secure connections (HTTP)
      keepConnection : Bool;   // Keep connection established after execution of request
      timeOut : Time := T#10s;   // Time to wait for response from server
   END_VAR
   VAR_OUTPUT
      connected : Bool;   // Connection to web server is established
      done : Bool;   // HTTP request finished
      busy : Bool;   // Function is busy
      error : Bool;   // An error occured
      status : Word := 16#7000;   // Specifies the error
      diagnostics : "typeDiagnostics";   // Diagnostics information of FB
      responseCode : UInt;   // HTTP response code
      length : UDInt;   // Length of received data
   END_VAR
   VAR_IN_OUT
      responseData : Array[*] of Char;   // Data received from HTTP server
   END_VAR
   VAR
      instTSendC : TSEND_C;   // Instance of TSEND_C
      instTRcv : TRCV;   // Instance of TRCV
      instTimeout : TON_TIME;   // Time-out
      statConnected : Bool;   // Static value for output 'connected'
      statDone : Bool;   // Static value for output 'done'
      statBusy : Bool;   // Static value for output 'busy'
      statError : Bool;   // Static value for output 'error'
      statStatus : Word := 16#7000;   // Static value for output 'status'
      statResponseCode : UInt;   // Static value for output 'responseCode'
      statLength : UDInt;   // Static value for output 'length'
      statFBState : USInt := 0;   // Current state in state machine
      statSubfunctionStatus : DWord;   // Status or return value of called FBs, FCs and system blocks
      statEmptyDiagnostics : "typeDiagnostics";   // Empty diagnostics information (for initialization purposes only)
      statParam : Struct   // Connection parameters
         isQDN : Bool;
         paramQDN : TCON_QDN_SEC;   // Connection parameters in form of QDN
         paramIP : TCON_IP_V4_SEC;   // Connection parameters in form of IP address
      END_STRUCT;
      statHost : String;   // Host part of URL
      statRequest : Struct   // GET request
         chars : Array[0..#UPPER_REQUEST_ARRAY] of Char;   // GET request (max. length: url (254) + data (254) + header (94)
         length : UInt;   // Length of GET request
      END_STRUCT;
      statSend : Struct   // Parameters for instruction TSend_C
         connect : Bool;   // Establish and keep connection
         req : Bool;   // Send data
      END_STRUCT;
      statEncoding : String;   // Transfer encoding of response from HTTP server
      statContentLength : UDInt;   // Content length as specified in header of response
      statChunkLen : UDInt;   // Remaining length of current chunk
      statRcvdLen : UDInt;   // Sum length of received data
      statTimeoutIn : Bool;   // Timeout
      statRcvBuffer : Array[0..#UPPER_TCP_FRAME] of Char;   // Temporary receive buffer
      statSizeRcvArray : UDInt;   // Size of receive buffer at parameter "responseData"
      statExecuteOld : Bool;   // Last cycle's value of input "execute"
      statHeaderComplete : Bool;   // Header was received completely
   END_VAR
   VAR_TEMP
      tempUrl : String;   // Copy of URL
      tempQuery : String;   // Query part of URL
      tempIndex : DInt;   // Index for for loops
      tempPos : Int;   // General tag for positions
      tempLen : UInt;   // General tag for lengths
      tempRet : Word;   // General tag for return values
      tempString : String;   // General tag for strings
      tempExitLoop : Bool;   // Condition to exit REPEAT loop around state machine
      tempChunk : Struct   // Temporary tags for chunked encoding
         posData : UInt;   // Start position of data in current packet
         lenData : UInt;   // Length of data in current packet
         exitLoop : Bool;   // Condition to exit loop
      END_STRUCT;
   END_VAR
   VAR CONSTANT
      UPPER_REQUEST_ARRAY : UInt := 1459;   // Upper limit of request array
      UPPER_TCP_FRAME : UInt := 1459;   // Upper limit of a TCP/IP frame
      UPPER_USER_FIELDS : USInt := 255;   // Upper limit of userFields
      PORT_UNSECURE : UInt := 80;   // Port for unsecure HTTP connection
      PORT_SECURE : UInt := 443;   // Port for secure HTTP connection
      POS_RESPONSE_CODE : USInt := 9;   // Position of HTTP response code in response message
      STATUS_DONE : Word := 16#0000;   // Job finished without errors
      STATUS_DISCONNECTED : Word := 16#0003;   // Communication connection closed
      STATUS_IDLE : Word := 16#7000;   // No job
      STATUS_FIRST_CALL : Word := 16#7001;   // First call after incoming new job (rising edge 'execute')
      STATUS_CONNECTING : Word := 16#7002;   // Connection is currently being established
      STATUS_DISCONNECTING : Word := 16#7003;   // Communication connection is being terminated
      STATUS_MONITORING : Word := 16#7004;   // Communication connection has been established and is being monitored. No send job execution active
      STATUS_SENT : Word := 16#7005;   // Request sent, waiting for response
      SUB_STATUS_NO_ERROR : DWord := 16#0000_0000;   // No error occured in subfunction call
      ERR_BOUND_NOT_ZERO : Word := 16#8201;   // Lower bound of receive buffer is not 0
      ERR_INVALID_URL : Word := 16#8202;   // Invalid URL
      ERR_DIFFERENT_HOST : Word := 16#8203;   // Trying to use existing connection with different host
      ERR_END_USER_FIELDS : Word := 16#8206;   // End of user-defined header fields could not be found
      ERR_REQUEST_SIZE : Word := 16#8210;   // Request array is too small for specified parameters
      ERR_RESPONSE_SIZE : Word := 16#8220;   // Receive buffer at parameter "responseData" too small
      ERR_CONN_LOST : Word := 16#8400;   // Offset for lost connection
      ERR_FORWARDING : Word := 16#8403;   // Server responded with forwarding message. Forwarding is not supported, see "diagnostics"
      ERR_WEBSERVER : Word := 16#8404;   // Webserver responded with error code, see "diagnostics"
      ERR_INVALID_HEADER : Word := 16#8405;   // Header of response is invalid or incomplete / Header of response is invalid
      ERR_TIMEOUT : Word := 16#8408;   // Time-out occurred
      ERR_UNDEFINED_STATE : Word := 16#8600;   // Error due to an undefined state in state machine
      ERR_TSENDC : Word := 16#8601;   // Error: TCON encountered an error, see "diagnostics"
      ERR_TRCV : Word := 16#8603;   // Error: TURCV encountered error, see "diagnostics"
      ERR_MOVE_USER_FIELDS : Word := 16#8612;   // Error in MOVE_BLK_VARIANT to copy user-defined header fields, see "diagnostics"
      ERR_ENCODING_UNKNOWN : Word := 16#8620;   // Transfer encoding of response could not be detected or is unsupported
      ERR_MOVE_IDENTITY : Word := 16#8630;   // Error in MOVE_BLK_VARIANT for transfer encoding 'identity', see "diagnostics"
      ERR_DECODING_FAILED : Word := 16#8640;   // Chunk encoded response could not be decoded
      ERR_MOVE_CHUNKED : Word := 16#8641;   // Error in MOVE_BLK_VARIANT for transfer encoding 'chunked', see "diagnostics"
      TSENDC_STATUS_CONNECTED : Word := 16#0001;   // TSEND_C: Communication connection established
      MOVE_STATUS_SIZE : Word := 16#8483;   // MOVE_BLK_VARIANT: DEST too small
      FB_STATE_NO_PROCESSING : USInt := 0;   // FB state: No processing
      FB_STATE_INIT : USInt := 1;   // FB state: initialization
      FB_STATE_REQUEST : USInt := 2;   // FB state: prepare request
      FB_STATE_SEND : USInt := 3;   // FB state: send request
      FB_STATE_RCV : USInt := 4;   // FB state: receive data
      FB_STATE_MON : USInt := 5;   // FB state: monitoring connection
      CRLF : String := '$R$L';   // Newline control character (carriage return, line feed)
      HEADER_END : String := '$R$L$R$L';   // End of HTTP header (two newline control characters)
      LEN_CRLF : UInt := 2;   // Length of CRLF
      SCHEME_HTTP : String := 'http://';   // Scheme HTTP
      SCHEME_HTTPS : String := 'https://';   // Scheme HTTPS
   END_VAR
   // statParam.paramIP.ConnPara.ActiveEstablished := true;
   // statParam.paramQDN.ConnPara.ActiveEstablished := true;
BEGIN
   REGION BLOCK INFO HEADER
     //===============================================================================
     // SIEMENS / (c)Copyright 2024
     //-------------------------------------------------------------------------------
     // Title:        LHTTP_Get
     // Function:     Implements the HTTP GET method
     // Library:      LHTTP
     // Author:       Siemens Industry Online Support
     // Tested with:  CPU 1516-3 PN/DP V2.9
     // Engineering:  TIA Portal V17
     // Restrictions: --
     // Requirements: S7-1200 with firmware V4.4 or higher
     //               S7-1500 with firmware V2.0 or higher
     //-------------------------------------------------------------------------------
     // Change log table:
     // Version  | Date       | Expert in charge       | Changes applied
     //----------|------------|------------------------|------------------------------
     // 02.02.00 | 2024-04-05 | Online Support         | Changed behavior that HTTPS is used by default
     //          |            |                        | Improved evaluation of host in URL
     //----------|------------|------------------------|------------------------------
     // 02.01.04 | 2023-08-23 | Online Support         | Fixed issue when first packet of response only contains header or response header is not received completely in one packet
     //----------|------------|------------------------|------------------------------
     // 02.01.01 | 2023-02-23 | Online Support         | Changed data type of "statContentLength" to allow larger content size
     //----------|------------|------------------------|------------------------------
     // 02.01.00 | 2021-12-15 | Online Support         | Renamed parameter "data" to "queryParams"
     //-------------------------------------------------------------------------------
     // 02.00.04 | 2021-05-10 | Online Support         | Fixed issues with chunked encoding
     //          |            |                        | Allow chunk sizes > 65535 Bytes
     //          |            |                        | Made header evaluation case-insensitive
     //-------------------------------------------------------------------------------
     // 02.00.00 | 2020-12-16 | Online Support         | Added option to keep connection established
     //          |            |                        | Added parameter to add user-defined headers fields
     //          |            |                        | Changed to data type of "data" to Variant to allow larger data
     //          |            |                        | Removed "statusID" and added "diagnostics" instead, changed some error codes
     //-------------------------------------------------------------------------------
     // 01.00.00 | 2019-04-01 | Online Support         | First released version
     //===============================================================================
   END_REGION

   REGION INSTRUCTIONS
     IF (#statStatus <> #STATUS_IDLE) THEN // Only execute when FB is triggered to reduce system load
       // Connect and send
       IF #statParam.isQDN THEN // Call if host is a domain name
         #instTSendC(REQ     := #statSend.req,
                     CONT    := #statSend.connect,
                     LEN     := #statRequest.length,
                     CONNECT := #statParam.paramQDN,
                     DATA    := #statRequest.chars);
       ELSE // Call if host is an IP address
         #instTSendC(REQ     := #statSend.req,
                     CONT    := #statSend.connect,
                     LEN     := #statRequest.length,
                     CONNECT := #statParam.paramIP,
                     DATA    := #statRequest.chars);
       END_IF;

       // Receive
       #instTRcv(ID    := #statParam.paramQDN.ConnPara.ID,
                 EN_R  := #statFBState >= #FB_STATE_RCV,
                 LEN   := 0,
                 ADHOC := true,
                 DATA  := #statRcvBuffer);

       // Monitor time out
       #instTimeout(IN := #statTimeoutIn,
                    PT := #timeOut);

       IF #instTimeout.Q THEN
         #statStatus := #ERR_TIMEOUT;
       END_IF;
     END_IF;
   END_REGION

   REGION TRIGGERING
     IF (#execute = true AND #statExecuteOld = false) // Check if FB is triggered
       AND (#statStatus = #STATUS_IDLE OR #statStatus = #STATUS_MONITORING)
     THEN // First call; initialize FB
       // Copy URL
       #tempUrl := #url;

       #statBusy := true;
       #statStatus := #STATUS_FIRST_CALL;
       #statSubfunctionStatus := #SUB_STATUS_NO_ERROR;
       #diagnostics := #statEmptyDiagnostics;

       IF #statConnected = FALSE THEN // Connection is not yet established
         #statFBState := #FB_STATE_INIT;
       ELSE // Connection is already established, skip init
         #statFBState := #FB_STATE_REQUEST;
       END_IF;

     ELSIF (#statStatus = #STATUS_FIRST_CALL) THEN
       #statStatus := #STATUS_CONNECTING;
     END_IF;

     // Edge detection 'execute' input
     #statExecuteOld := #execute;
   END_REGION TRIGGERING

   IF (#statStatus = #STATUS_IDLE) THEN // Nothing to do -> End here to reduce "system load"
     RETURN;
   END_IF;

   REGION STATE_MACHINE
     // State machine is wrapped in REPEAT loop to make it possible to quickly exit state machine
     // in case of an error or to go through CASE multiple times within one cycle
     REPEAT
       #tempExitLoop := true; // Condition to exit loop is set per default

       CASE #statFBState OF // State machine of FB
         #FB_STATE_NO_PROCESSING: // No processing active
           ;

         #FB_STATE_INIT:
           REGION INIT
             // Get size of receive buffer
             IF LOWER_BOUND(ARR := #responseData, DIM := 1) <> 0 THEN
               #statStatus := #ERR_BOUND_NOT_ZERO;
               EXIT;
             ELSE
               #statSizeRcvArray := DINT_TO_UDINT(UPPER_BOUND(ARR := #responseData, DIM := 1)) + 1;
             END_IF;

             // Set connection parameters
             #statParam.paramQDN.ConnPara.InterfaceId := #hwID;
             #statParam.paramQDN.ConnPara.ID := #connID;
             #statParam.paramIP.ConnPara.InterfaceId := #hwID;
             #statParam.paramIP.ConnPara.ID := #connID;

             // Check if 'http' was explicitely specified for connection to be unsecure
             IF LEFT(IN := #tempUrl, L := LEN(#SCHEME_HTTP)) = #SCHEME_HTTP THEN // HTTP
               #statParam.paramQDN.ActivateSecureConn := false;
               #statParam.paramIP.ActivateSecureConn := false;
               #tempUrl := DELETE(IN := #tempUrl, L := LEN(#SCHEME_HTTP), P := 1); // Delete network protocol from URL
             ELSE // HTTPS
               #statParam.paramQDN.ActivateSecureConn := true;
               #statParam.paramQDN.ExtTLSCapabilities.%X0 := #tls.validateServerIdentity;
               #statParam.paramQDN.TLSServerCertRef := #tls.serverCert;
               #statParam.paramQDN.TLSClientCertRef := #tls.clientCert;
               #statParam.paramIP.ActivateSecureConn := true;
               #statParam.paramIP.ExtTLSCapabilities.%X0 := #tls.validateServerIdentity;
               #statParam.paramIP.TLSServerCertRef := #tls.serverCert;
               #statParam.paramIP.TLSClientCertRef := #tls.clientCert;

               // Delete network protocol from URL if specified
               IF LEFT(IN := #tempUrl, L := LEN(#SCHEME_HTTPS)) = #SCHEME_HTTPS THEN
                 #tempUrl := DELETE(IN := #tempUrl, L := LEN(#SCHEME_HTTPS), P := 1);
               END_IF;
             END_IF;

             // Get host name and port
             #tempPos := FIND(IN1 := #tempUrl, IN2 := '/');
             IF #tempPos > 0 THEN // URL has a path after host name
               #statHost := LEFT(IN := #tempUrl, L := #tempPos - 1); // Strip path
             ELSE
               #statHost := #tempUrl;
             END_IF;

             #tempPos := FIND(IN1 := #statHost, IN2 := ':');
             IF #tempPos > 0 THEN // Port specified in URL
               #statParam.paramQDN.ConnPara.RemotePort := STRING_TO_UINT(DELETE(IN := #statHost, L := #tempPos, P := 1));
               #statParam.paramIP.ConnPara.RemotePort := STRING_TO_UINT(DELETE(IN := #statHost, L := #tempPos, P := 1));
               #statHost := LEFT(IN := #statHost, L := #tempPos - 1); // Strip port
             ELSE // No port specified in URL, set default port
               IF #statParam.paramQDN.ActivateSecureConn OR #statParam.paramIP.ActivateSecureConn THEN
                 #statParam.paramQDN.ConnPara.RemotePort := #PORT_SECURE;
                 #statParam.paramIP.ConnPara.RemotePort := #PORT_SECURE;
               ELSE
                 #statParam.paramQDN.ConnPara.RemotePort := #PORT_UNSECURE;
                 #statParam.paramIP.ConnPara.RemotePort := #PORT_UNSECURE;
               END_IF;
             END_IF;

             // Determine if host is domain name or IP address
             #statParam.isQDN := NOT "IsIPAddress"(address := #statHost, ipAddress => #statParam.paramIP.ConnPara.RemoteAddress);

             IF #statParam.isQDN THEN // Host is a domain name
               #statParam.paramQDN.ConnPara.RemoteQDN := CONCAT(IN1 := #statHost, IN2 := '.');
             END_IF;

             #statFBState := #FB_STATE_REQUEST;
             #tempExitLoop := FALSE; // Don't exit loop to go directly to prepare request
           END_REGION INIT

         #FB_STATE_REQUEST:
           REGION PREP_REQUEST
             // Check host in URL when using existing connection
             IF #statConnected = TRUE THEN
               #tempPos := FIND(IN1 := #tempUrl, IN2 := #statHost);
               IF #tempPos = 0 THEN // URL doesn't contain expected host
                 #statStatus := #ERR_DIFFERENT_HOST;
                 EXIT;
               ELSE // Scheme and host must be deleted for further processing
                 #tempUrl := DELETE(IN := #tempUrl, L := #tempPos + LEN(#statHost) - 1, P := 1);
               END_IF;
             END_IF;

             // Get path
             #tempPos := FIND(IN1 := #tempUrl, IN2 := '/');
             IF #tempPos > 0 THEN // URL has a path after host name
               #tempString := DELETE(IN := #tempUrl, L := #tempPos - 1, P := 1);
             ELSE
               #tempString := '/';
             END_IF;

             // Prepare query part of URL
             IF #queryParams <> '' THEN // Parameter is in use
               IF #queryParams[1] = '?' OR #queryParams[1] = '&' THEN
                 #tempQuery := DELETE(IN := #queryParams, P := 1, L := 1);
               ELSE
                 #tempQuery := #queryParams;
               END_IF;
               #tempPos := FIND(IN1 := #tempString, IN2 := '?'); // Check if URL already contains query parameters
               IF #tempPos <> 0 THEN // URL already contains query parameters
                 #tempQuery := CONCAT(IN1 := '&', IN2 := #tempQuery); // Append query parameters with &
               ELSE // URL does not contain query parameters
                 #tempQuery := CONCAT(IN1 := '?', IN2 := #tempQuery); // Append query parameters with ?
               END_IF;
             END_IF;

             // Put together GET request
             // Strg_TO_Chars conversion is done several times to utilize maximum length of parameters url and query parameters
             Strg_TO_Chars(Strg   := CONCAT(IN1 := 'GET ', IN2 := #tempString), // Path cannot be longer than 249 characters --> save to use CONCAT
                           pChars := 0,
                           Cnt    => #tempLen,
                           Chars  := #statRequest.chars);
             #tempPos := UINT_TO_INT(#tempLen);

             Strg_TO_Chars(Strg   := #tempQuery,
                           pChars := #tempPos,
                           Cnt    => #tempLen,
                           Chars  := #statRequest.chars);
             #tempPos += UINT_TO_INT(#tempLen);

             Strg_TO_Chars(Strg   := CONCAT(IN1 := ' HTTP/1.1$R$LHost: ', IN2 := #statHost), // Host will not use all 254 characters --> save to use CONCAT
                           pChars := #tempPos,
                           Cnt    => #tempLen,
                           Chars  := #statRequest.chars);
             #tempPos += UINT_TO_INT(#tempLen);

             Strg_TO_Chars(Strg   := '$R$LUser-Agent: SIMATIC Controller (LHTTP)$R$LAccept: text/html$R$LAccept-Encoding: identity$R$LAccept-Charset: utf-8$R$L',
                           pChars := #tempPos,
                           Cnt    => #tempLen,
                           Chars  := #statRequest.chars);
             #tempPos += UINT_TO_INT(#tempLen);

             // Insert additional user-defined header fields
             IF #userFields[0] <> ' ' THEN
               FOR #tempLen := 0 TO #UPPER_USER_FIELDS DO
                 IF #userFields[#tempLen] = '$00' THEN
                   EXIT;
                 END_IF;
               END_FOR;

               IF #tempLen > #UPPER_USER_FIELDS THEN // End not found
                 #statStatus := #ERR_END_USER_FIELDS;
                 EXIT;
               END_IF;

               #tempRet := INT_TO_WORD(MOVE_BLK_VARIANT(SRC := #userFields, COUNT := #tempLen, SRC_INDEX := 0, DEST_INDEX := #tempPos, DEST => #statRequest.chars));

               IF #tempRet = #MOVE_STATUS_SIZE THEN
                 #statStatus := #ERR_REQUEST_SIZE;
                 EXIT;
               ELSIF #tempRet <> 16#0000 THEN
                 #statStatus := #ERR_MOVE_USER_FIELDS;
                 #statSubfunctionStatus := #tempRet;
                 EXIT;
               END_IF;

               #tempPos += UINT_TO_INT(#tempLen);

               // Append CRLF if needed
               IF #statRequest.chars[#tempPos - 2] <> '$R' AND #statRequest.chars[#tempPos - 1] <> '$L' THEN
                 #statRequest.chars[#tempPos] := '$R';
                 #statRequest.chars[#tempPos + 1] := '$L';
                 #tempPos += 2;
               END_IF;
             END_IF;

             // Append end of header section
             Strg_TO_Chars(Strg   := #CRLF,
                           pChars := #tempPos,
                           Cnt    => #tempLen,
                           Chars  := #statRequest.chars);
             #tempPos += UINT_TO_INT(#tempLen);

             // Calculate total length of request
             #statRequest.length := INT_TO_UINT(#tempPos);

             #statSend.connect := true; // Connect
             #statSend.req := true; // Send request
             #statTimeoutIn := true; // Start timer
             #statFBState := #FB_STATE_SEND;
           END_REGION

         #FB_STATE_SEND: // Send data
           REGION SEND
             IF #instTSendC.STATUS = #TSENDC_STATUS_CONNECTED THEN
               #statConnected := TRUE;
             ELSIF #instTSendC.DONE THEN
               #statStatus := #STATUS_SENT;
               #statFBState := #FB_STATE_RCV;
               // Don't exit loop to go directly to receive state
               // without waiting for next cycle so that no responses can be missed
               #tempExitLoop := false;
             ELSIF #instTSendC.ERROR THEN
               #statStatus := #ERR_TSENDC;
               #statSubfunctionStatus := #instTSendC.STATUS;
             END_IF;
           END_REGION

         #FB_STATE_RCV: // Wait for new data
           REGION RCV
             IF #instTRcv.NDR AND #instTRcv.RCVD_LEN > 0 THEN

               REGION HEADER_EVAL
                 // Evaluate header
                 IF NOT #statHeaderComplete THEN

                   REGION response code
                     IF #statResponseCode = 0 THEN // First packet
                       // Get response code
                       Chars_TO_Strg(Chars  := #statRcvBuffer,
                                     pChars := #POS_RESPONSE_CODE,
                                     Cnt    := 3,
                                     Strg   => #tempString);
                       #statResponseCode := STRING_TO_UINT(#tempString);

                       // Exit loop immediately and output errror if response code shows errors or forwarding
                       IF #statResponseCode >= 300 THEN
                         #tempRet := ATH(IN := #tempString, N := 3, OUT => #statSubfunctionStatus); // Interpret response code as hexadecimal
                         #statSubfunctionStatus := SHR(IN := #statSubfunctionStatus, N := 20);
                         IF #statResponseCode >= 400 THEN
                           #statStatus := #ERR_WEBSERVER;
                         ELSE
                           #statStatus := #ERR_FORWARDING;
                         END_IF;
                         EXIT; // Exit loop immediately and output errror 
                       END_IF;
                     END_IF;
                   END_REGION response code

                   REGION transfer encoding
                     // Search header for content length
                     #tempRet := "LHTTP_ExtractStringFromArray"(textBefore := 'Content-Length: ',
                                                                textAfter := #CRLF,
                                                                extractedString => #tempString,
                                                                searchIn := #statRcvBuffer);

                     IF #tempRet <> 0 THEN // Content length not found; try lower-case
                       #tempRet := "LHTTP_ExtractStringFromArray"(textBefore := 'content-length: ',
                                                                  textAfter := #CRLF,
                                                                  extractedString => #tempString,
                                                                  searchIn := #statRcvBuffer);
                     END_IF;

                     IF #tempRet = 0 THEN // Content length found
                       #statContentLength := STRING_TO_UDINT(#tempString);
                       #statEncoding := 'identity';
                     ELSE // Can't detect content length, check if transfer encoding is 'chunked'
                       #tempPos := DINT_TO_INT("LHTTP_FindStringInArray"(searchFor := 'chunked', searchIn := #statRcvBuffer));

                       IF #tempPos >= 0 THEN
                         #statEncoding := 'chunked';
                       END_IF;
                     END_IF;
                   END_REGION transfer encoding

                   REGION header end
                     // Find header end
                     #tempPos := DINT_TO_INT("LHTTP_FindStringInArray"(searchFor := #HEADER_END, searchIn := #statRcvBuffer));

                     IF #tempPos > 0 THEN // Header end found
                       #statHeaderComplete := TRUE;
                       #tempPos += LEN(#HEADER_END); // Beginning of content

                       IF #statEncoding = '' THEN // Header end found but encoding not detected
                         #statStatus := #ERR_ENCODING_UNKNOWN;
                         EXIT;
                       END_IF;

                       IF #instTRcv.RCVD_LEN = #tempPos THEN // Packet contains no body, wait for next packet
                         EXIT;
                       END_IF;

                     ELSE // Header incomplete, wait for next packet
                       EXIT;
                     END_IF;
                   END_REGION header end
                 END_IF;
               END_REGION

               REGION TE_IDENTITY
                 IF #statEncoding = 'identity' THEN // Transfer encoding is 'identity'
                   // Move data from buffer to output; tempLen contains header length during first packet, otherwise 0
                   #tempRet := INT_TO_WORD(MOVE_BLK_VARIANT(SRC := #statRcvBuffer,
                                                                                    COUNT := MIN(IN1 := #instTRcv.RCVD_LEN - INT_TO_UDINT(#tempPos), IN2 := #statSizeRcvArray - #statRcvdLen), // Move as much as possible to output
                                                                                    SRC_INDEX := #tempPos,
                                                                                    DEST_INDEX := UDINT_TO_DINT(#statRcvdLen),
                                                                                    DEST => #responseData));

                   // Exit loop immediately and output error if data could not be moved
                   IF #tempRet <> 0 THEN
                     #statStatus := #ERR_MOVE_IDENTITY;
                     #statSubfunctionStatus := #tempRet;
                     EXIT;
                   END_IF;

                   // Add length of received packet to sum; tempPos contains position of beginning of content
                   #statRcvdLen += #instTRcv.RCVD_LEN - INT_TO_UDINT(#tempPos);

                   IF #statRcvdLen > #statSizeRcvArray THEN // Receive buffer too small
                     #statStatus := #ERR_RESPONSE_SIZE;
                     #statLength := #statContentLength; // Output required size of buffer
                   ELSIF #statRcvdLen >= #statContentLength THEN // Everything was received
                     #statStatus := #STATUS_DONE;
                     #statLength := #statRcvdLen;
                   END_IF;
                 END_IF;
               END_REGION

               REGION TE_CHUNKED
                 IF #statEncoding = 'chunked' THEN // Transfer encoding is 'chunked'

                   // Set position of chunk data
                   #tempChunk.posData := INT_TO_UINT(#tempPos); // tempPos contains position of beginning of content

                   REPEAT
                     #tempChunk.exitLoop := true; // Condition to exit loop is set per default

                     // Read length of chunk if received packet is first packet or a previous chunk was received completely
                     IF #statChunkLen = 0 THEN
                       // Extract hexadecimal chunk-size field
                       Chars_TO_Strg(Chars  := #statRcvBuffer,
                                     pChars := #tempChunk.posData,
                                     Cnt    := 0,
                                     Strg   => #tempString);
                       #tempPos := FIND(IN1 := #tempString, IN2 := #CRLF);
                       #tempRet := ATH(IN := #tempString, N := #tempPos - 1, OUT => #statChunkLen);
                       // Shift bits to the right depending on length of chunk size, since ATH is left aligned
                       #statChunkLen := SHR(IN := #statChunkLen, N := 4 * INT_TO_UINT(8 - (#tempPos - 1)));

                       // Move start position of data behind chunk-size field
                       #tempChunk.posData += INT_TO_UINT(#tempPos) + 1;

                       // Exit loop immediately and output error if chunk size cannot be detected
                       IF #tempRet <> 0 THEN
                         #statStatus := #ERR_DECODING_FAILED;
                         EXIT;
                       END_IF;
                     END_IF;

                     IF #statChunkLen = 0 THEN // Length was evaluated, chunk contains no data --> final chunk received
                       #statStatus := #STATUS_DONE;
                       #statLength := #statRcvdLen;
                     ELSE // Chunk contains data
                       // Evaluate length of received packet and set length of data accordingly
                       IF #instTRcv.RCVD_LEN = #tempChunk.posData + #statChunkLen + #LEN_CRLF THEN // Chunk was received entirely and packet contains no further chunks
                         #tempChunk.lenData := UDINT_TO_UINT(#statChunkLen); // Output remaining length of chunk
                       ELSIF #instTRcv.RCVD_LEN < #tempChunk.posData + #statChunkLen + #LEN_CRLF THEN // Packet only contains part of chunk
                         #tempChunk.lenData := UDINT_TO_UINT(#instTRcv.RCVD_LEN) - #tempChunk.posData; // Output entire packet without possible chunk-size field
                       ELSIF #instTRcv.RCVD_LEN > #tempChunk.posData + #statChunkLen + #LEN_CRLF THEN // Current packet contains more than one chunk
                         #tempChunk.lenData := UDINT_TO_UINT(#statChunkLen); // Output remaining length of chunk
                         #tempChunk.exitLoop := false; // Execute loop again since packet contains more data
                       ELSE // Can't decode message
                         #statStatus := #ERR_DECODING_FAILED;
                         EXIT;
                       END_IF;

                       // Move received data to output
                       #tempRet := INT_TO_WORD(MOVE_BLK_VARIANT(SRC := #statRcvBuffer,
                                                                                        COUNT := MIN(IN1 := #tempChunk.lenData, IN2 := #statSizeRcvArray - #statRcvdLen), // Move as much as possible to output
                                                                                        SRC_INDEX := #tempChunk.posData,
                                                                                        DEST_INDEX := UDINT_TO_DINT(#statRcvdLen),
                                                                                        DEST => #responseData));

                       // Exit loop immediately and output error if data could not be moved
                       IF #tempRet <> 0 THEN
                         #statStatus := #ERR_MOVE_CHUNKED;
                         #statSubfunctionStatus := #tempRet;
                         EXIT;
                       END_IF;

                       // Move start position of data behind data of current chunk in case packet contains more data; only relevant if REPEAT loop is executed again
                       #tempChunk.posData += #tempChunk.lenData + #LEN_CRLF;

                       // Subtract length of data in current packet from remaining length of chunk and add to sum of received data
                       #statChunkLen -= #tempChunk.lenData;
                       #statRcvdLen += #tempChunk.lenData;

                       IF #statRcvdLen > #statSizeRcvArray THEN // Receive buffer too small
                         #statStatus := #ERR_RESPONSE_SIZE;
                         #statLength := #statRcvdLen; // Output required size of buffer according to so far received chunked messages
                         EXIT;
                       END_IF;
                     END_IF;
                   UNTIL (#tempChunk.exitLoop = true) END_REPEAT;
                 END_IF;
               END_REGION

             ELSIF #instTRcv.ERROR THEN
               #statStatus := #ERR_TRCV;
               #statSubfunctionStatus := #instTRcv.STATUS;
             END_IF;
           END_REGION

         #FB_STATE_MON:
           REGION MONITORING
             IF #keepConnection = FALSE THEN // Trigger to disconnect
               #statSend.connect := FALSE;
               #statDone := FALSE;
               #statBusy := TRUE;
               #statStatus := #STATUS_DISCONNECTING;
             END_IF;

             IF #instTSendC.STATUS = #STATUS_DISCONNECTED THEN
               #statConnected := FALSE;
               #statStatus := #STATUS_DISCONNECTED;
             ELSIF #instTRcv.ERROR THEN
               #statConnected := FALSE;
               #statStatus := #ERR_CONN_LOST OR (#instTRcv.STATUS AND 16#00FF);
             END_IF;
           END_REGION

         ELSE // Undefined state in state machine reached
           #statStatus := #ERR_UNDEFINED_STATE;
       END_CASE;

     UNTIL (#tempExitLoop = true) END_REPEAT;
   END_REGION

   REGION OUTPUTS
     // Write outputs
     IF (#statStatus = #STATUS_DONE) AND (#statDone = false) THEN // Execution finished without errors
       #statDone := true;
       #statBusy := false;
       #statError := false;
       #statSend.connect := #keepConnection;
       #statSend.req := false;
       #statTimeoutIn := false;

       IF #keepConnection THEN
         // execution finished but connection is kept alive --> set state monitoring
         #statFBState := #FB_STATE_MON;
       ELSE
         #statConnected := FALSE;
         // execution finished --> set state no processing
         #statFBState := #FB_STATE_NO_PROCESSING;
       END_IF;

     ELSIF (#statStatus = #STATUS_DISCONNECTED) AND (#statBusy = true) THEN // Connection was terminated separately of send job
       #statConnected := FALSE;
       #statBusy := FALSE;
       // execution finished --> set state no processing
       #statFBState := #FB_STATE_NO_PROCESSING;

     ELSIF (#statStatus.%X15 = true) AND (#statError = false) THEN // Error occurred (#statStatus is 16#8000 to 16#FFFF)
       #statConnected := false;
       #statDone := false;
       #statBusy := false;
       #statError := true;
       #statSend.connect := false; // After error, connection is always terminated
       #statSend.req := false;
       #statTimeoutIn := false;
       // Write diagnostics
       #diagnostics.status := #statStatus;
       #diagnostics.subfunctionStatus := #statSubfunctionStatus;
       #diagnostics.stateNumber := #statFBState;
       // execution aborted --> set state no processing
       #statFBState := #FB_STATE_NO_PROCESSING;

     ELSIF ((#execute = false) AND ((#statDone = true) OR (#statError = true)))
       OR ((#statStatus = #STATUS_DISCONNECTED) AND (#statBusy = false)) // Connection was terminated separately of send job
     THEN // Reset outputs
       #statDone := false;
       #statBusy := false;
       #statError := false;
       #statResponseCode := 0;
       #statLength := 0;
       #statHeaderComplete := FALSE;
       #statContentLength := 0;
       #statChunkLen := 0;
       #statEncoding := '';
       #statRcvdLen := 0;

       IF #statConnected THEN
         #statStatus := #STATUS_MONITORING;
       ELSE
         #statStatus := #STATUS_IDLE;
       END_IF;
     END_IF;

     // Write static values to outputs
     #connected := #statConnected;
     #done := #statDone;
     #busy := #statBusy;
     #error := #statError;
     #status := #statStatus;
     #responseCode := #statResponseCode;
     #length := #statLength;
     ENO := NOT #statError;
   END_REGION OUTPUTS
END_FUNCTION_BLOCK

